{attribute 'qualified_only'}
{attribute 'strict'}
{attribute 'to_string'}
TYPE E_DemoStep :
(
	ManualMode := -1, // "Do nothing" used to interact with MC3 Motion UI
	Init := 0,
	WaitForIO,
	DetectMovers,
	SortMovers,	
	Enabling,
	SquareUpMovers,
	MoveToSeqenceStartPos,
	JoinTrack,
	FigureEight,
	LeaveTrack,
	GoToOpositeCorner,
	FlyBy,
	MoveAroundPerimeter,
	MoveToCenterOfTiles,
	RotateInverse,
	Spin,
	Lift,
	Tilt,
	Disable
) := ManualMode;
END_TYPE

(* stored: Version 1.1.0.1, ProductVersion 3.1.4026.20
   DUT E_DemoStep: Id {ec2e79b1-db13-496a-827a-4cb926db1174} *)
